# B&R Automation Studio project DancerControl
Automation Studio 4.12.6.106; technology packages: Acp10Arnc0 5.26.1

## Configuration Config1

CPU X20CP1586, AutomationRuntime J4.93, Build 4.1.2, Vc V4.73.2

### Task classes (Cpu.sw)
```
Cyclic#4:
  VMaster <- Axis.VMaster.prg
NcDataObjects: acp10etxen <- Axis.AxisObject.acp10etxen.dob, AxInit <- Axis.AxisObject.RealAxis.AxInit.dob, AcpParTab <- Axis.AxisObject.RealAxis.AcpParTab.dob, VAxInit <- Axis.AxisObject.Virtual.VAxInit.dob
Libraries: Acp10man, Acp10par, NcGlobal, Acp10sim, Acp10_MC, sys_lib, brsystem, runtime, MpAxis, MpBase, MpCom, MTWinder, MTTypes, AsBrMath
```

### Hardware
```
8EIxxxHxD1x.xxxx-1 : 8EIxxxHxD1x.xxxx-1 v2.3.1.1  [PLK1 -> X20CP1586.IF3 (NodeNumber=1) [Cable Type=PowerlinkCable, Length=10, Version=1.0.0.3]]
  MotionTP = Acp10Arnc0
  Simulate = complete
  ActiveMotorSimulation_r1 = on
  BothEndSwitchesAreNormallyOpen_r1 = on
  QuickStopIsNormallyOpen_r1 = on
  ActiveMotorSimulation_r2 = on
  BothEndSwitchesAreNormallyOpen_r2 = on
  QuickStopIsNormallyOpen_r2 = on
X20CP1586 : X20CP1586 v1.10.0.0
  Connector IF2:
    ActivateDevice = 1
  ConfigurationID = DancerControl_Config1
  Simulation = 1
  TimerDeviceType = EPLX2X
  TimerDevice = X20CP1586.IF3
  TaskClassIdleTime = 2000
  FileDevice1
  FileDeviceName1 = USER
  FileDevicePath1 = USER_PATH
```

### Acp10cfg.ncc - X20CP1586/Motion/Acp10cfg.ncc
```
NcConfiguration (Version=5.26.1, NcSwId=Acp10)
  ACP10CF1_typ:
    cnt_nettrc_rec_drive = 1500
    bufsize_trace_upload = 1200
    tc_nc_man_task = Cyclic #1
    glob_pv_as_ncobject = Yes
    ncsys_dl_broadcast = Yes
    ncsys_dl_acp_reset = Yes
    safemc_log_err_to_ax = Yes
    network_init:
      ncsw_init_execute = Yes
      automatic_execute = No
      node_nr_warning = Yes
      net_err_before_ncact = Yes
    nettrc:
      enter_parsecrec = Yes
      enter_ncaction = Yes
      save_ring_startidx = Yes
    cam_prof_download:
      cam_dat_dl_parallel = No
      tc_cam_dl_parallel = Task class for NC Manager task
    plk_if[0]:
      if_name = IF3
      tc_CycDat_PLCopen = Task class for NC Manager task
      mc_broadcast_extdat = No
```

### Acp10map.ncm - X20CP1586/Motion/Acp10map.ncm
```
NcMapping (NcSwId=Acp10, DisabledNodesAreHidden=False)
  NcObject gAxReelA (ModuleId=8EIxxxHxD1x.xxxx-1, Type=ncAXIS, Channel=1, AcoposSimulation=Off, InitParameter=AxInit, AcoposParameter=AcpParTab, Disabled=FALSE, ModuleDisabled=FALSE)
  NcObject gAxReelB (ModuleId=8EIxxxHxD1x.xxxx-1, Type=ncAXIS, Channel=2, AcoposSimulation=Off, InitParameter=AxInit, AcoposParameter=AcpParTab, Disabled=FALSE, ModuleDisabled=FALSE)
  NcObject gVMaster (ModuleId=8EIxxxHxD1x.xxxx-1, Type=ncV_AXIS, Channel=1, InitParameter=VAxInit, Disabled=FALSE, ModuleDisabled=FALSE)
  NcObject 8EIxxxHxD1x.xxxx-1_ncV_AXIS2 (ModuleId=8EIxxxHxD1x.xxxx-1, Type=ncV_AXIS, Channel=2, Disabled=TRUE, ModuleDisabled=FALSE)
```

### Config.mpaxisbasic - X20CP1586/Motion/Config.mpaxisbasic
```
Element gVMasterLink (Type=mpaxisbasic)
  AxisConfiguration = AxisWithConfiguration
    Drive:
      Controller:
        LoopFilters:
          [0]
          [1]
          [2]
Element gReelALink (Type=mpaxisbasic)
  AxisConfiguration = AxisWithConfiguration
    Drive:
      Controller:
        LoopFilters:
          [0]
          [1]
          [2]
Element gReelBLink (Type=mpaxisbasic)
  AxisConfiguration = AxisWithConfiguration
    Drive:
      Controller:
        LoopFilters:
          [0]
          [1]
          [2]
```

## Logical view

Binary libraries used (declarations not repeated): operator, runtime, astime, AsIecCon, Acp10man 5.26.1, Acp10par 5.26.1, NcGlobal 5.26.1, Acp10sim 5.26.1, Acp10_MC 5.26.1, sys_lib, brsystem, MpAxis 1.89.0, MpBase, MpCom 5.24.2, MTWinder, MTTypes, AsBrMath

### Global.typ - Global data types
```iecst
TYPE
	axis_command_typ : 	STRUCT  (*command structure*)
		Power : BOOL; (*switch on the controller*)
		Home : BOOL; (*reference the axis*)
		MoveAbsolute : BOOL; (*move to an defined position*)
		MoveAdditive : BOOL; (*move a defiened distance*)
		MoveVelocity : BOOL; (*start a movement with a defiened velocity*)
		Halt : BOOL; (*stop every active movement*)
		Stop : BOOL; (*stop every active movement as long as is set*)
		MoveJogPos : BOOL; (*move in positive direction as long as is set*)
		MoveJogNeg : BOOL; (*move in negative direction as long as is set*)
		ErrorAcknowledge : BOOL; (*reset active errors*)
		VelocityControl : BOOL; (*activate velocity control*)
	END_STRUCT;
	axis_parameter_typ : 	STRUCT  (*parameter structure*)
		Position : REAL; (*target-position for MoveAbsolute-Command*)
		Distance : REAL; (*distance for MoveAdditive-Command*)
		Velocity : REAL; (*velocity for MoveVelocity-Command*)
		Direction : USINT; (*direction for commanded movements*)
		Acceleration : REAL; (*acceleration for commanded movements*)
		Deceleration : REAL; (*deceleration for commanded movements*)
		HomePosition : REAL; (*target-position for referencing the axis*)
		HomeMode : USINT; (*homing mode*)
		JogVelocity : REAL; (*velocity for jogging movement*)
	END_STRUCT;
	axis_status_typ : 	STRUCT  (*status structure*)
		ErrorID : UINT; (*ErrorID of any occured error*)
		ErrorText : ARRAY[0..3]OF STRING[79]; (*Error Text*)
		ActPosition : REAL; (*actual position of the axis*)
		ActVelocity : REAL; (*actual velocity of the axis*)
		DriveStatus : MpAxisBasicInfoType; (*actual status of the axis*)
		PoweredOn : BOOL; (*Axis powered on *)
		Homed : BOOL; (*Axis Homed*)
	END_STRUCT;
	axis_axisState_typ : 	STRUCT  (*axis state structure*)
		Disabled : BOOL; (*if set, axis is in state Disabled*)
		StandStill : BOOL; (*if set, axis is in state StandsStill*)
		Homing : BOOL; (*if set, axis is in state Homing*)
		Stopping : BOOL; (*if set, axis is in state Stopping*)
		DiscreteMotion : BOOL; (*if set, axis is in state DiscreteMotion*)
		ContinuousMotion : BOOL; (*if set, axis is in state ContinousMotion*)
		SynchronizedMotion : BOOL; (*if set, axis is in state SynchronizedMotion*)
		ErrorStop : BOOL; (*if set, axis is in state ErrorStop*)
	END_STRUCT;
	axis_typ : 	STRUCT  (*control structure*)
		Command : axis_command_typ; (*command structure*)
		Parameter : axis_parameter_typ; (*parameter structure*)
		Status : axis_status_typ; (*status structure*)
		AxisState : axis_axisState_typ; (*axis state structure*)
		Enable : BOOL; (*Axis command enable*)
	END_STRUCT;

END_TYPE
```

### Global.var - Global variables
```iecst
(*Axis Structure *)
VAR
	gAxReelA : ACP10AXIS_typ;
	gAxReelB : ACP10AXIS_typ;
	gVMaster : ACP10VAXIS_typ;
END_VAR
(*Control Axis Structure *)
VAR
	gAxis : ARRAY[0..MAX_AXIS] OF axis_typ;
	AxisIndex : USINT;
END_VAR
```

### Constants.var
```iecst
VAR CONSTANT
	MAX_AXIS : USINT := 3; (*Max value axis to be controlled *)
END_VAR
(*Axis Identifier*)
VAR CONSTANT
	VMASTER : USINT := 0;
	REEL_A : USINT := 1;
	REEL_B : USINT := 2;
	GENERIC : USINT := 3;
END_VAR
(*Axis Parameters*)
VAR CONSTANT
	LINE_ACCELERATION : REAL := 500000.0; (*Acceleration and deceleration of the line axis.*)
	MAX_LINE_DECELERATION : REAL := 1000000.0; (*Maximum deceleration of the line axis.*)
	MAX_DANCER_POSITION : REAL := 500.0; (*Maximum position of the dancer arm.*)
	STANDSTILL_WINDOW : REAL := 0.0; (*Speed dead band*)
	PI : REAL := 3.1416; (*PI Value*)
END_VAR
```


### Program Logical/Axis/VMaster (IEC)

#### Cyclic.st - Cyclic code
```iecst
PROGRAM _CYCLIC

	(**** Call Subroutines ****)
	Act_Main;
	Act_Parameters;

	(** Enable FB's **)
	AxisBasic.Enable 			:= gAxis[AxisIndex].Enable;
	AxisConfig.Enable 		:= AxisBasic.Active;
	ReadAxisError.Enable 	:= AxisBasic.Error OR AxisConfig.Error;

	(**** Definicion sentido de giro del eje ****)
	IF AxisDirection THEN
		Direction	:= mpAXIS_DIR_CLOCKWISE;
	ELSE
		Direction	:= mpAXIS_DIR_COUNTERCLOCKWISE;
	END_IF

	(**** Secuencia configuarcion Eje *****)
	IF NOT ConfigReq THEN
		StConfig := CONFIG_WAIT;
	END_IF

	CASE StConfig OF

		CONFIG_WAIT:

			IF ConfigReq THEN
				StConfig := CONFIG_LOAD_REQ;
			END_IF

		CONFIG_LOAD_REQ:

			(* Carga la configuracion por default en Confing.mpaxisbasic*)
			AxisConfig.Load	:= TRUE;

			IF AxisConfig.CommandDone THEN
				StConfig 			:= CONFIG_LOAD_DONE;
			END_IF

		CONFIG_LOAD_DONE:

			(* Actualiza la configuracion, carga parametros asignados por el usuario *)
			AxisConfig.Load		:= FALSE;
			StConfig 					:= CONFIG_SAVE_REQ;

		CONFIG_SAVE_REQ:

			AxisConfigPar.AxisName 																:= AxisName;

			//Axis

			AxisConfigPar.Axis.BaseType 													:= mpAXIS_PERIODIC_ROTARY;
			AxisConfigPar.Axis.MeasurementUnit 										:= mpAXIS_UNIT_GENERIC;
			AxisConfigPar.Axis.MeasurementResolution 							:= Resolution;
			AxisConfigPar.Axis.PeriodSettings.Period							:= Period;

			AxisConfigPar.Axis.MovementLimits.VelocityPositive		:= LimitSpeed;
			AxisConfigPar.Axis.MovementLimits.VelocityNegative		:= LimitSpeed;
			AxisConfigPar.Axis.MovementLimits.Acceleration				:= LimitAccDec;
			AxisConfigPar.Axis.MovementLimits.Deceleration				:= LimitAccDec;

			//Drive

			AxisConfigPar.Drive.Gearbox.Input											:= GearIn;
			AxisConfigPar.Drive.Gearbox.Output										:= GearOut;
			AxisConfigPar.Drive.Gearbox.Direction 								:= Direction;
			AxisConfigPar.Drive.Transformation.ReferenceDistance 	:= Period;

			(* Salva en el drive los parametros asignados por el usuario *)

			AxisConfig.Save := TRUE;

			IF AxisConfig.CommandDone THEN
				StConfig := CONFIG_SAVE_DONE;
			END_IF

		CONFIG_SAVE_DONE:

			(* Configuracion terminada *)

			AxisConfig.Save := FALSE;
			ConfigReq				:= FALSE;
			ConfigDone			:= TRUE;

	END_CASE

	(********** FB's Configuration *********)

	AxisBasic.Axis 					:= Axis;
	AxisBasic.MpLink 				:= ADR(MpLink);
	AxisBasic.Parameters 		:= ADR(AxisBasicPar);
	AxisBasic();

	AxisConfig.MpLink 			:= ADR(MpLink);
	AxisConfig.Configuration:= ADR(AxisConfigPar);
	AxisConfig();

	ReadAxisError.Axis 			:= Axis;
	ReadAxisError.Mode 			:= mcTEXT;
	ReadAxisError();

	(****************************************)

END_PROGRAM
```

#### Act_Main.st
```iecst
ACTION Act_Main:

	(*Command*)
	gAxis[AxisIndex].Command.Power := AxisBasic.Active AND AxisConfig.Active;
	AxisBasic.Stop := gAxis[AxisIndex].Command.Stop;

	(*Status*)
	gAxis[AxisIndex].Status.ActVelocity := AxisBasic.Velocity;
	gAxis[AxisIndex].Status.ActPosition := LREAL_TO_REAL(AxisBasic.Position);
	gAxis[AxisIndex].Status.PoweredOn 	:= AxisBasic.PowerOn;
	gAxis[AxisIndex].Status.Homed				:= AxisBasic.IsHomed;
	gAxis[AxisIndex].Status.DriveStatus.PLCopenState := AxisBasic.Info.PLCopenState;
	gAxis[AxisIndex].Status.PoweredOn 	:= AxisBasic.PowerOn;

	(*Axis State*)
	gAxis[AxisIndex].AxisState.Disabled 	:= NOT AxisBasic.Active;
	gAxis[AxisIndex].AxisState.StandStill := NOT AxisBasic.MoveActive;
	gAxis[AxisIndex].AxisState.ErrorStop 	:= AxisBasic.Error OR AxisConfig.Error;
	gAxis[AxisIndex].AxisState.StandStill := NOT AxisBasic.MoveActive;
	gAxis[AxisIndex].AxisState.ErrorStop 	:= AxisBasic.Error OR AxisConfig.Error;

	(*Error Reset*)
	IF gAxis[AxisIndex].Command.ErrorAcknowledge THEN
		AxisBasic.ErrorReset := TRUE;
		AxisConfig.ErrorReset := TRUE;
	ELSE
		AxisBasic.ErrorReset := FALSE;
		AxisConfig.ErrorReset := FALSE;
	END_IF

	(**** Configuracion FB Read Axis Error ****)
	ReadAxisError.Configuration.Format 					:= mcWRAP;   //ReadAxisErrorPar;
	ReadAxisError.Configuration.LineLength 			:= SIZEOF(gAxis[AxisIndex].Status.ErrorText[0]);
	ReadAxisError.Configuration.DataLength 			:= SIZEOF(gAxis[AxisIndex].Status.ErrorText);
	ReadAxisError.Configuration.DataAddress 		:= ADR(gAxis[AxisIndex].Status.ErrorText[0]);
	ReadAxisError.Configuration.DataObjectName 	:= 'acp10etxen';

	(**** Error ****)

	IF gAxis[AxisIndex].AxisState.ErrorStop THEN
		StAxis := STATE_ERROR;
	END_IF

	(**** Speed Control/Accel Control ****)

	AxisBasicPar.Velocity 		:= gAxis[AxisIndex].Parameter.Velocity;
	AxisBasicPar.Acceleration	:= gAxis[AxisIndex].Parameter.Acceleration;
	AxisBasicPar.Deceleration := gAxis[AxisIndex].Parameter.Deceleration;

	IF OldVelocity <> AxisBasicPar.Velocity OR OldAccel <> AxisBasicPar.Acceleration OR OldDecel <> AxisBasicPar.Deceleration THEN
		AxisBasic.Update := TRUE;
		OldVelocity := AxisBasicPar.Velocity;
		OldAccel := AxisBasicPar.Acceleration;
		OldDecel := AxisBasicPar.Deceleration;
	ELSE
		AxisBasic.Update := FALSE;
	END_IF

	(**** Checks is the motor is powered On ****)

	IF NOT gAxis[AxisIndex].Command.Power THEN
		StAxis := STATE_WAIT;
	END_IF

	(**** Axis Sequencer ****)

	CASE StAxis OF

		STATE_WAIT:

			IF AxisBasic.Active AND AxisBasic.Info.BootState = mpAXIS_BLP_DONE AND AxisBasic.Info.ReadyToPowerOn AND ConfigDone THEN
				StAxis:= STATE_POWER_ON;
			ELSIF gAxis[AxisIndex].Command.Power AND NOT ConfigDone THEN
				ConfigReq:= TRUE;
			END_IF

		STATE_POWER_ON:

			IF AxisBasic.Info.HardwareInfo.DeviceType = mpAXIS_VIRTUAL THEN
				StAxis:= STATE_HOME;
			END_IF

		STATE_HOME:

			IF NOT AxisBasic.IsHomed THEN
				AxisBasic.Home := TRUE;
			ELSIF AxisBasic.IsHomed THEN
				AxisBasic.Home := FALSE;
				StAxis:= STATE_READY;
			END_IF

		STATE_READY:

			IF gAxis[AxisIndex].Command.MoveVelocity THEN
				StAxis:= STATE_AUTO;
			END_IF

		STATE_AUTO:

			AxisBasic.MoveVelocity := TRUE;

			IF NOT gAxis[AxisIndex].Command.MoveVelocity THEN
				AxisBasic.MoveVelocity := FALSE;
				StAxis:= STATE_STOP;
			END_IF

		STATE_STOP:

			AxisBasic.Stop := TRUE;

			IF AxisBasic.Stopped THEN
				AxisBasic.Stop := FALSE;
				StAxis:= STATE_READY;
			END_IF

		STATE_ERROR :

			AxisBasic.MoveVelocity := FALSE;

			IF gAxis[AxisIndex].Command.ErrorAcknowledge THEN
				StAxis:= STATE_READY;
			END_IF

	END_CASE

	gAxis[AxisIndex].AxisState.ContinuousMotion := StAxis = STATE_AUTO;
	gAxis[AxisIndex].AxisState.Stopping 				:= StAxis = STATE_STOP;
	gAxis[AxisIndex].AxisState.StandStill 			:= StAxis = STATE_READY;

END_ACTION
```

#### Act_Parameters.st
```iecst
ACTION Act_Parameters:

	//---- Numero del Eje ----///
	AxisIndex := VMASTER;

	//---- MpLink ----//
	MpLink 		:= gVMasterLink;
	Axis 			:= ADR(gVMaster);

	//---- Nombre del eje ----//
	AxisName := ' Virtual Master ';

	//---- Hablita el eje ----//
	gAxis[AxisIndex].Enable := TRUE;

	//---- Limite de velocidad -----//
	LimitSpeed 	:= 6600.0;

	//----- Limete de aceleracion/desaceleracion ----//
	LimitAccDec := 6600.0;

	//---- Relacion de velocoidad motor/reductor ----//
	GearIn 	:= 1;
	GearOut := 1;

	//---- Seleccion direccion de rotacion del eje ----//
	AxisDirection := TRUE; // TRUE = sentido de las manesillas del reloj; FALSE = en contra de las manesillas del reloj;

	// ---- Definicion Paramentros de posicion del eje ----//
	Period 				:= 360.0;
	Resolution		:= 0.01;

	/////////////////////////////////////////////////////////////////

END_ACTION
```

#### Init.st - Init code
```iecst
PROGRAM _INIT

	ConfigReq := TRUE;
	Act_Parameters;

END_PROGRAM
```

#### Types.typ - Local data types
```iecst
TYPE
	AxisState_enum :
		( (*Axis control steps*)
		STATE_WAIT := 0,
		STATE_POWER_ON := 10,
		STATE_ERROR := 20,
		STATE_STOP := 30,
		STATE_READY := 40,
		STATE_HOME := 50,
		STATE_AUTO := 60,
		STATE_MANUAL := 70,
		STATE_MAINT := 80
		);
	ConfigStates_enum :
		( (*Axis Configuration steps *)
		CONFIG_WAIT := 0,
		CONFIG_LOAD_REQ := 10,
		CONFIG_LOAD_DONE := 20,
		CONFIG_SAVE_REQ := 30,
		CONFIG_SAVE_DONE := 70,
		CONFIG_COMPLETE := 80
		);
END_TYPE
```

#### Variables.var - Local variables
```iecst
	(*Mp Axis FB*)
VAR
		AxisBasic : MpAxisBasic;
		AxisBasicPar : MpAxisBasicParType;
		AxisConfig : MpAxisBasicConfig;
		AxisConfigPar : MpAxisBasicConfigType;
		ReadAxisError : MC_BR_ReadAxisError;
END_VAR
	(*Axis Control Var *)
	VAR
		Axis : UDINT; (*Axis*)
		AxisIndex : USINT; (*Axis Index *)
		StAxis : AxisState_enum; (*Axis control steps*)
		MpLink : MpComIdentType; (*Axis basic parameters structure*)
END_VAR
	(*Axis Speed Control var *)
	VAR
		OldVelocity : REAL; (*Old Velocity Value*)
END_VAR
	(*Axis Configuration*)
	VAR
		StConfig : ConfigStates_enum; (*Configuration steps*)
		ConfigDone : BOOL; (*Configuration done*)
		AxisDirection : BOOL; (*Command direction 1 = CW; 0 = CCW*)
		Direction : MpAxisMotorDirectionEnum; (*Status diection *)
		ConfigReq : BOOL; (*Configuration command*)
		LimitSpeed : REAL; (*Speed limmit*)
		LimitAccDec : REAL; (*acceleratio/Deceleration limit*)
		GearIn : UDINT; (*Input ratio*)
		GearOut : UDINT; (*output ratio*)
		Period : LREAL; (*Period  exemple 360.0 degrees.*)
		Resolution : REAL; (*Minimum distance that can be used for a movement*)
		AxisName : STRING[20]; (*Axis Name *)
		OldAccel : REAL; (*Old Acel value *)
		OldDecel : REAL; (*Old  decel value*)
END_VAR
```

### Data object Logical/Axis/AxisObject/acp10etxen (Ett)

- acp10etxen.ett (not shown)

### Program Logical/Axis/ReelA

#### Types.typ
```iecst
TYPE
	AxisState_enum :
		( (*Axis control steps*)
		STATE_WAIT := 0,
		STATE_POWER_ON := 10,
		STATE_ERROR := 20,
		STATE_STOP := 30,
		STATE_READY := 40,
		STATE_HOME := 50,
		STATE_AUTO := 60,
		STATE_MANUAL := 70,
		STATE_MAINT := 80
	);
	ConfigStates_enum :
		( (*Axis Configuration steps *)
		CONFIG_WAIT := 0,
		CONFIG_LOAD_REQ := 10,
		CONFIG_LOAD_DONE := 20,
		CONFIG_SAVE_REQ := 30,
		CONFIG_SAVE_DONE := 70
	);

END_TYPE
```

#### Variables.var
```iecst
VAR
	(*Mp Axis FB*)
	AxisBasic : MpAxisBasic;
	AxisBasicPar : MpAxisBasicParType;
	AxisConfig : MpAxisBasicConfig;
	AxisConfigPar : MpAxisBasicConfigType;
	ReadAxisError : MC_BR_ReadAxisError;
	VelocityControl : MC_BR_VelocityControl; (*Function Block*)
END_VAR
(*Axis Control Var *)
VAR
	Axis : UDINT;(*Axis*)
	AxisIndex : USINT; (*Axis Index *)
	StAxis : AxisState_enum; (*Axis control steps*)
	MpLink : MpComIdentType;  (*Axis basic parameters structure*)
END_VAR
(*Axis Speed Control var *)
VAR
	OldVelocity : REAL; (*Old Velocity Value*)
END_VAR
(*Axis Configuration*)
VAR
	StConfig : ConfigStates_enum; (*Configuration steps*)
	ConfigDone : BOOL;(*Configuration done*)
	AxisDirection : BOOL; (*Command direction 1 = CW; 0 = CCW*)
	Direction : MpAxisMotorDirectionEnum; (*Status diection *)
	ConfigReq : BOOL; (*Configuration command*)
	LimitSpeed : REAL;(*Speed limmit*)
	LimitAccDec : REAL;(*acceleratio/Deceleration limit*)
	GearIn : UDINT;
	GearOut : UDINT;
	Period : LREAL;
	Resolution : REAL;
	AxisName : STRING[20];
END_VAR
```

#### Act_Main.st
```iecst
ACTION Act_Main:

	(*Command*)
	gAxis[AxisIndex].Command.Power := AxisBasic.Active AND AxisConfig.Active;
	AxisBasic.Stop := gAxis[AxisIndex].Command.Stop;

	(*Status*)
	gAxis[AxisIndex].Status.ActVelocity := AxisBasic.Velocity;
	gAxis[AxisIndex].Status.ActPosition := LREAL_TO_REAL(AxisBasic.Position);
	gAxis[AxisIndex].Status.PoweredOn 	:= AxisBasic.PowerOn;
	gAxis[AxisIndex].Status.Homed				:= AxisBasic.IsHomed;
	gAxis[AxisIndex].Status.DriveStatus.PLCopenState := AxisBasic.Info.PLCopenState;
	gAxis[AxisIndex].Status.PoweredOn 	:= AxisBasic.PowerOn;

	(*Axis State*)
	gAxis[AxisIndex].AxisState.Disabled 	:= NOT AxisBasic.Active;
	gAxis[AxisIndex].AxisState.StandStill := NOT AxisBasic.MoveActive;
	gAxis[AxisIndex].AxisState.ErrorStop 	:= AxisBasic.Error OR AxisConfig.Error;
	gAxis[AxisIndex].AxisState.StandStill := NOT AxisBasic.MoveActive;
	gAxis[AxisIndex].AxisState.ErrorStop 	:= AxisBasic.Error OR AxisConfig.Error;

	(*Error Reset*)
	IF gAxis[AxisIndex].Command.ErrorAcknowledge THEN
		AxisBasic.ErrorReset := TRUE;
		AxisConfig.ErrorReset := TRUE;
	ELSE
		AxisBasic.ErrorReset := FALSE;
		AxisConfig.ErrorReset := FALSE;
	END_IF

	(**** Configuracion FB Read Axis Error ****)
	ReadAxisError.Configuration.Format 					:= mcWRAP;   //ReadAxisErrorPar;
	ReadAxisError.Configuration.LineLength 			:= SIZEOF(gAxis[AxisIndex].Status.ErrorText[0]);
	ReadAxisError.Configuration.DataLength 			:= SIZEOF(gAxis[AxisIndex].Status.ErrorText);
	ReadAxisError.Configuration.DataAddress 		:= ADR(gAxis[AxisIndex].Status.ErrorText[0]);
	ReadAxisError.Configuration.DataObjectName 	:= 'acp10etxen';

	(**** Error ****)

	IF gAxis[AxisIndex].AxisState.ErrorStop THEN
		StAxis := STATE_ERROR;
	END_IF

//	(**** Speed Control/Accel Control ****)
//
//	AxisBasicPar.Velocity 		:= gAxis[AxisIndex].Parameter.Velocity;
//	AxisBasicPar.Acceleration	:= gAxis[AxisIndex].Parameter.Acceleration;
//	AxisBasicPar.Deceleration := gAxis[AxisIndex].Parameter.Deceleration;
//
//	IF OldVelocity <> AxisBasicPar.Velocity OR OldAccel <> AxisBasicPar.Acceleration OR OldDecel <> AxisBasicPar.Deceleration THEN
//		AxisBasic.Update := TRUE;
//		OldVelocity := AxisBasicPar.Velocity;
//		OldAccel := AxisBasicPar.Acceleration;
//		OldDecel := AxisBasicPar.Deceleration;
//	ELSE
//		AxisBasic.Update := FALSE;
//	END_IF

	(**** Checks is the motor is powered On ****)

	IF NOT gAxis[AxisIndex].Command.Power THEN
		StAxis := STATE_WAIT;
	END_IF

	(**** Checks the motor error ****)

	IF gAxis[AxisIndex].AxisState.ErrorStop THEN
		StAxis:= STATE_ERROR;
	END_IF

	(**** Axis Sequencer ****)

	CASE StAxis OF

		STATE_WAIT:

			IF AxisBasic.Active AND AxisBasic.Info.BootState = mpAXIS_BLP_DONE AND AxisConfig.Active AND AxisBasic.Info.ReadyToPowerOn AND ConfigDone THEN
				StAxis:= STATE_POWER_ON;
			ELSIF gAxis[AxisIndex].Command.Power AND NOT ConfigDone THEN
				ConfigReq:= TRUE;
			END_IF

		STATE_POWER_ON:

			IF gAxis[AxisIndex].Command.Power AND NOT AxisBasic.PowerOn THEN
				AxisBasic.Power := TRUE;
			ELSIF AxisBasic.PowerOn THEN
				StAxis:= STATE_HOME;
			END_IF

		STATE_HOME:

			IF NOT AxisBasic.IsHomed THEN
				AxisBasic.Home := TRUE;
			ELSIF AxisBasic.IsHomed THEN
				AxisBasic.Home := FALSE;
				StAxis:= STATE_READY;
			END_IF

		STATE_READY:

			IF gAxis[AxisIndex].Command.VelocityControl THEN
				StAxis:= STATE_AUTO;
			END_IF

		STATE_AUTO:

			(******************** VELOCITY CONTROL **********************)
			(* STATE: velocity control *)
			(* activate MC_BR_VelocityControl *)
						VelocityControl.Enable := TRUE;
						VelocityControl.CyclicVelocity := gSetWinderVelocity;
						VelocityControl.CyclicVelocityCorrection :=  gVelocityCorrection;
						VelocityControl.CyclicTorque := gSetMotorTorque;
						VelocityControl.Acceleration := gAxis[AxisIndex].Parameter.Acceleration;
						VelocityControl.Deceleration := gAxis[AxisIndex].Parameter.Deceleration ;
						VelocityControl.TorqueMode := mcFF;
						VelocityControl.SctrlKv := gActProportionalGain;
						VelocityControl.SctrlTn := gActIntegrationTime;
			(* this feature is not possible for ACOPOS simulation *)
			// VelocityControl.InitSctrl := gControl.Winder.InitSpeedController;

			IF NOT gAxis[AxisIndex].Command.VelocityControl THEN
				VelocityControl.Enable := FALSE;
				StAxis:= STATE_READY;
			END_IF

		STATE_ERROR:

			VelocityControl.Enable := FALSE;

	END_CASE

END_ACTION
```

#### Act_Parameters.st
```iecst
ACTION Act_Parameters:

	//---- Numero del Eje ----///
	AxisIndex := REEL_A;

	//---- MpLink ----//
	MpLink 		:= gReelALink;
	Axis 			:= ADR(gAxReelA);

	//---- Nombre del eje ----//
	AxisName := ' Reel A ';

	//---- Hablita el eje ----//
	gAxis[AxisIndex].Enable := TRUE;

	//---- Limite de velocidad -----//
	LimitSpeed 	:= 6600.0;

	//----- Limete de aceleracion/desaceleracion ----//
	LimitAccDec := 6600.0;

	//---- Relacion de velocoidad motor/reductor ----//
	GearIn 	:= 1;
	GearOut := 1;

	//---- Seleccion direccion de rotacion del eje ----//
	AxisDirection := TRUE; // TRUE = sentido de las manesillas del reloj; FALSE = en contra de las manesillas del reloj;

	// ---- Definicion Paramentros de posicion del eje ----//
	Period 				:= 360.0;
	Resolution		:= 0.001;

	/////////////////////////////////////////////////////////////////

END_ACTION
```

#### Cyclic.st
```iecst
PROGRAM _CYCLIC

(**** Call Subroutines ****)
	Act_Main;
	Act_Parameters;

	(** Enable FB's **)
	AxisBasic.Enable 			:= gAxis[AxisIndex].Enable;
	AxisConfig.Enable 		:= AxisBasic.Active;
	ReadAxisError.Enable 	:= AxisBasic.Error OR AxisConfig.Error;

	(**** Definicion sentido de giro del eje ****)
	IF AxisDirection THEN
		Direction	:= mpAXIS_DIR_CLOCKWISE;
	ELSE
		Direction	:= mpAXIS_DIR_COUNTERCLOCKWISE;
	END_IF

	(**** Secuencia configuarcion Eje *****)
	IF NOT ConfigReq THEN
		StConfig := CONFIG_WAIT;
	END_IF

	CASE StConfig OF

		CONFIG_WAIT:

			IF ConfigReq THEN
				StConfig := CONFIG_LOAD_REQ;
			END_IF

		CONFIG_LOAD_REQ:

			(* Carga la configuracion por default en Confing.mpaxisbasic*)
			AxisConfig.Load	:= TRUE;

			IF AxisConfig.CommandDone THEN
				StConfig 			:= CONFIG_LOAD_DONE;
			END_IF

		CONFIG_LOAD_DONE:

			(* Actualiza la configuracion, carga parametros asignados por el usuario *)
			AxisConfig.Load		:= FALSE;
			StConfig 					:= CONFIG_SAVE_REQ;

		CONFIG_SAVE_REQ:

			AxisConfigPar.AxisName 																:= AxisName;

			//Axis

			AxisConfigPar.Axis.BaseType 													:= mpAXIS_PERIODIC_ROTARY;
			AxisConfigPar.Axis.MeasurementUnit 										:= mpAXIS_UNIT_GENERIC;
			AxisConfigPar.Axis.MeasurementResolution 							:= Resolution;
			AxisConfigPar.Axis.PeriodSettings.Period							:= Period;

			AxisConfigPar.Axis.MovementLimits.VelocityPositive		:= LimitSpeed;
			AxisConfigPar.Axis.MovementLimits.VelocityNegative		:= LimitSpeed;
			AxisConfigPar.Axis.MovementLimits.Acceleration				:= LimitAccDec;
			AxisConfigPar.Axis.MovementLimits.Deceleration				:= LimitAccDec;

			//Drive

			AxisConfigPar.Drive.Gearbox.Input											:= GearIn;
			AxisConfigPar.Drive.Gearbox.Output										:= GearOut;
			AxisConfigPar.Drive.Gearbox.Direction 								:= Direction;
			AxisConfigPar.Drive.Transformation.ReferenceDistance 	:= Period;

			(* Salva en el drive los parametros asignados por el usuario *)

			AxisConfig.Save := TRUE;

			IF AxisConfig.CommandDone THEN
				StConfig := CONFIG_SAVE_DONE;
			END_IF

		CONFIG_SAVE_DONE:

			(* Configuracion terminada *)

			AxisConfig.Save := FALSE;
			ConfigReq				:= FALSE;
			ConfigDone			:= TRUE;

	END_CASE

	(********** FB's Configuration *********)

	AxisBasic.Axis 					:= Axis;
	AxisBasic.MpLink 				:= ADR(MpLink);
	AxisBasic.Parameters 		:= ADR(AxisBasicPar);
	AxisBasic();

	AxisConfig.MpLink 			:= ADR(MpLink);
	AxisConfig.Configuration:= ADR(AxisConfigPar);
	AxisConfig();

	ReadAxisError.Axis 			:= Axis;
	ReadAxisError.Mode 			:= mcTEXT;
	ReadAxisError();

	VelocityControl();
	(****************************************)

END_PROGRAM
```

### Program Logical/Axis/ReelB

#### Types.typ
```iecst
TYPE
	AxisState_enum :
		( (*Axis control steps*)
		STATE_WAIT := 0,
		STATE_POWER_ON := 10,
		STATE_ERROR := 20,
		STATE_STOP := 30,
		STATE_READY := 40,
		STATE_HOME := 50,
		STATE_AUTO := 60,
		STATE_MANUAL := 70,
		STATE_MAINT := 80
	);
	ConfigStates_enum :
		( (*Axis Configuration steps *)
		CONFIG_WAIT := 0,
		CONFIG_LOAD_REQ := 10,
		CONFIG_LOAD_DONE := 20,
		CONFIG_SAVE_REQ := 30,
		CONFIG_SAVE_DONE := 70
	);
END_TYPE
```

#### Variables.var
```iecst
VAR
	(*Mp Axis FB*)
	AxisBasic : MpAxisBasic;
	AxisBasicPar : MpAxisBasicParType;
	AxisConfig : MpAxisBasicConfig;
	AxisConfigPar : MpAxisBasicConfigType;
	ReadAxisError : MC_BR_ReadAxisError;
	VelocityControl : MC_BR_VelocityControl; (*Function Block*)
END_VAR
(*Axis Control Var *)
VAR
	Axis : UDINT;(*Axis*)
	AxisIndex : USINT; (*Axis Index *)
	StAxis : AxisState_enum; (*Axis control steps*)
	MpLink : MpComIdentType;  (*Axis basic parameters structure*)
END_VAR
(*Axis Speed Control var *)
VAR
	OldVelocity : REAL; (*Old Velocity Value*)
END_VAR
(*Axis Configuration*)
VAR
	StConfig : ConfigStates_enum; (*Configuration steps*)
	ConfigDone : BOOL;(*Configuration done*)
	AxisDirection : BOOL; (*Command direction 1 = CW; 0 = CCW*)
	Direction : MpAxisMotorDirectionEnum; (*Status diection *)
	ConfigReq : BOOL; (*Configuration command*)
	LimitSpeed : REAL;(*Speed limmit*)
	LimitAccDec : REAL;(*acceleratio/Deceleration limit*)
	GearIn : UDINT;
	GearOut : UDINT;
	Period : LREAL;
	Resolution : REAL;
	AxisName : STRING[20];
END_VAR
```

#### Act_Parameters.st
```iecst
ACTION Act_Parameters:

	//---- Numero del Eje ----///
	AxisIndex := REEL_B;

	//---- MpLink ----//
	MpLink 		:= gReelBLink;
	Axis 			:= ADR(gAxReelB);

	//---- Nombre del eje ----//
	AxisName := ' Reel A ';

	//---- Hablita el eje ----//
	gAxis[AxisIndex].Enable := TRUE;

	//---- Limite de velocidad -----//
	LimitSpeed 	:= 6600.0;

	//----- Limete de aceleracion/desaceleracion ----//
	LimitAccDec := 6600.0;

	//---- Relacion de velocoidad motor/reductor ----//
	GearIn 	:= 1;
	GearOut := 1;

	//---- Seleccion direccion de rotacion del eje ----//
	AxisDirection := TRUE; // TRUE = sentido de las manesillas del reloj; FALSE = en contra de las manesillas del reloj;

	// ---- Definicion Paramentros de posicion del eje ----//
	Period 				:= 360.0;
	Resolution		:= 0.001;

	/////////////////////////////////////////////////////////////////

END_ACTION
```

#### Cyclic.st
```iecst
PROGRAM _CYCLIC

	(**** Call Subroutines ****)
	Act_Main;
	Act_Parameters;

	(** Enable FB's **)
	AxisBasic.Enable 			:= gAxis[AxisIndex].Enable;
	AxisConfig.Enable 		:= AxisBasic.Active;
	ReadAxisError.Enable 	:= AxisBasic.Error OR AxisConfig.Error;

	(**** Definicion sentido de giro del eje ****)
	IF AxisDirection THEN
		Direction	:= mpAXIS_DIR_CLOCKWISE;
	ELSE
		Direction	:= mpAXIS_DIR_COUNTERCLOCKWISE;
	END_IF

	(**** Secuencia configuarcion Eje *****)
	IF NOT ConfigReq THEN
		StConfig := CONFIG_WAIT;
	END_IF

	CASE StConfig OF

		CONFIG_WAIT:

			IF ConfigReq THEN
				StConfig := CONFIG_LOAD_REQ;
			END_IF

		CONFIG_LOAD_REQ:

			(* Carga la configuracion por default en Confing.mpaxisbasic*)
			AxisConfig.Load	:= TRUE;

			IF AxisConfig.CommandDone THEN
				StConfig 			:= CONFIG_LOAD_DONE;
			END_IF

		CONFIG_LOAD_DONE:

			(* Actualiza la configuracion, carga parametros asignados por el usuario *)
			AxisConfig.Load		:= FALSE;
			StConfig 					:= CONFIG_SAVE_REQ;

		CONFIG_SAVE_REQ:

			AxisConfigPar.AxisName 																:= AxisName;

			//Axis

			AxisConfigPar.Axis.BaseType 													:= mpAXIS_PERIODIC_ROTARY;
			AxisConfigPar.Axis.MeasurementUnit 										:= mpAXIS_UNIT_GENERIC;
			AxisConfigPar.Axis.MeasurementResolution 							:= Resolution;
			AxisConfigPar.Axis.PeriodSettings.Period							:= Period;

			AxisConfigPar.Axis.MovementLimits.VelocityPositive		:= LimitSpeed;
			AxisConfigPar.Axis.MovementLimits.VelocityNegative		:= LimitSpeed;
			AxisConfigPar.Axis.MovementLimits.Acceleration				:= LimitAccDec;
			AxisConfigPar.Axis.MovementLimits.Deceleration				:= LimitAccDec;

			//Drive

			AxisConfigPar.Drive.Gearbox.Input											:= GearIn;
			AxisConfigPar.Drive.Gearbox.Output										:= GearOut;
			AxisConfigPar.Drive.Gearbox.Direction 								:= Direction;
			AxisConfigPar.Drive.Transformation.ReferenceDistance 	:= Period;

			(* Salva en el drive los parametros asignados por el usuario *)

			AxisConfig.Save := TRUE;

			IF AxisConfig.CommandDone THEN
				StConfig := CONFIG_SAVE_DONE;
			END_IF

		CONFIG_SAVE_DONE:

			(* Configuracion terminada *)

			AxisConfig.Save := FALSE;
			ConfigReq				:= FALSE;
			ConfigDone			:= TRUE;

	END_CASE

	(********** FB's Configuration *********)

	AxisBasic.Axis 					:= Axis;
	AxisBasic.MpLink 				:= ADR(MpLink);
	AxisBasic.Parameters 		:= ADR(AxisBasicPar);
	AxisBasic();

	AxisConfig.MpLink 			:= ADR(MpLink);
	AxisConfig.Configuration:= ADR(AxisConfigPar);
	AxisConfig();

	ReadAxisError.Axis 			:= Axis;
	ReadAxisError.Mode 			:= mcTEXT;
	ReadAxisError();

	VelocityControl();
	(****************************************)

END_PROGRAM
```

#### Init.st
```iecst
PROGRAM _INIT

	ConfigReq := TRUE;
	Act_Parameters;

END_PROGRAM
```

### Program Logical/DancerCtrl/LineCtrl (IEC)

#### Types.typ
```iecst
TYPE
	AxisState_enum :
		( (*States*)
		STATE_HOMING, (*Homing axis*)
		STATE_STANDSTILL, (*Axis ready*)
		STATE_MOTION, (*Continious movement*)
		STATE_STOPPING (*Stopping*)
	);
END_TYPE
```

#### Variables.var
```iecst
VAR
	RollerDiamter : REAL;
	LinearVelocity : REAL;
	AngularVelocity : REAL;
	Start : BOOL;
	StLineCtrl : AxisState_enum;
	Stop : BOOL;
END_VAR
```

#### Main.st
```iecst
PROGRAM _INIT

	(**** Datos de simulacion ****)
	RollerDiamter:= 100.0; // Diametro del rodillo en milimetros
	gAxis[VMASTER].Parameter.Acceleration := 10000.0; // grados/s
	gAxis[VMASTER].Parameter.Deceleration := 10000.0; // grados/s
	LinearVelocity := 400.0; // Setpoint en mm/s

END_PROGRAM

PROGRAM _CYCLIC

	(**** Calculo de velocidad para cambiarla a mm/s ****)
	gAxis[VMASTER].Parameter.Velocity := ((LinearVelocity * 360)/(PI * RollerDiamter));
	AngularVelocity := (gAxis[VMASTER].Status.ActVelocity * (PI/180)) * (RollerDiamter / 2);
	(*LinearVelocity := gControl.Cmd.LineVelocity;*)
	gLineVelocity :=  AngularVelocity/0.001;

	CASE StLineCtrl OF

		STATE_HOMING:

			(*************** STATE HOMING **************************)

			IF gAxis[VMASTER].Status.Homed THEN
				StLineCtrl:= STATE_STANDSTILL;
			END_IF

		STATE_STANDSTILL:

			(*************** STATE STANDSTILL **********************)

			IF Start THEN
				StLineCtrl := STATE_MOTION;
			END_IF

		STATE_MOTION:

			(*************** STATE MOTION **************************)

			(*gAxis[VMASTER].Parameter.Acceleration := 10000.0; // grados/s*)
			(*gAxis[VMASTER].Parameter.Deceleration := 10000.0; // grados/s*)

			Start := FALSE;
			gAxis[VMASTER].Command.MoveVelocity := TRUE;
			gAxis[REEL_A].Command.VelocityControl := TRUE;

			IF Stop THEN
				gAxis[VMASTER].Command.MoveVelocity := FALSE;
				gAxis[REEL_A].Command.VelocityControl := FALSE;
				StLineCtrl := STATE_STOPPING;
			END_IF

		STATE_STOPPING:

			(*************** STATE STOPPING ************************)

			Stop := FALSE;

			IF gAxis[VMASTER].Status.ActVelocity = 0.0 THEN
				StLineCtrl:= STATE_STANDSTILL;
			END_IF

	END_CASE

END_PROGRAM

PROGRAM _EXIT
	(* Insert code here *)

END_PROGRAM
```

### Program Logical/DancerCtrl/DancerController (IEC)

#### Cyclic.st - Cyclic code
```iecst
PROGRAM _CYCLIC

	Act_DiamEstimator;
	Act_Dancer;
	Act_SimModel;
	Act_AxisController;

END_PROGRAM
```

#### Act_DiamEstimator.st
```iecst
ACTION Act_DiamEstimator:

	DiameterEstimator.ActLinePosition := ActLinePosition;
	DiameterEstimator.ActWinderPosition := ActWinderPosition;
	DiameterEstimator.ActDancerPosition := ActDancerPosition;

	ActDiameter := DiameterEstimator.ActDiameter;

	(*************** DiameterEstimator ***********************)

	ActLinePosition		:= REAL_TO_DINT(gAxis[VMASTER].Status.ActPosition);
	ActWinderPosition := REAL_TO_DINT(gAxis[REEL_A].Status.ActPosition);

	DiameterEstimator();

END_ACTION
```

#### Act_Dancer.st
```iecst
ACTION Act_Dancer:

	DancerController.SetDancerPosition := SetDancerPosition;
	DancerController.ActDancerPosition := ActDancerPosition;

	DancerController.ActDiameter := ActDiameter;

	(*************** DancerController *************************)

	DancerController();

	VelocityCorrection := DancerController.VelocityCorrection;

	gVelocityCorrection := VelocityCorrection;

END_ACTION
```

#### Act_SimModel.st
```iecst
ACTION Act_SimModel:

	SimulationModel.Configuration := ConfigurationParameters;
	SimulationModel.Parameters := SimulationParameters;
	SimulationModel.SetLineVelocity := SetLineVelocity;

	SimulationModel.SetWinderVelocity := SetWinderVelocity;
	SimulationModel.WinderVelocityCorrection := WinderVelocityCorrection;
	SimulationModel.SetMotorTorque := SetMotorTorque;

	SimulationModel.ActProportionalGain := ActProportionalGain;
	SimulationModel.ActIntegrationTime := ActIntegrationTime;
	SimulationModel.InitSpeedController := InitSpeedController;

	(*************** SimulationModel **************************)

	SimulationModel();

END_ACTION
```

#### Act_AxisController.st
```iecst
ACTION Act_AxisController:

	SetLineVelocity := gLineVelocity; // Noe

	AxisController.SetLineVelocity  :=  SetLineVelocity;
	AxisController.ActDiameter  :=  ActDiameter;
	AxisController.SetMaterialTension  :=  SetMaterialTension;

	AxisController.SynchronizationTime  :=  SynchronistionTime;
	AxisController.StartSynchronization  :=  StartSynchronisation;
	AxisController.StopSynchronization  :=  StopSynchronisation;

	AxisController();

	SetWinderVelocity  :=  AxisController.SetWinderVelocity;
	SetMotorTorque  :=  AxisController.SetMotorTorque;

	ActProportionalGain  :=  AxisController.ActProportionalGain;
	ActIntegrationTime  :=  AxisController.ActIntegrationTime;
	InitSpeedController  :=  AxisController.InitSpeedController;

	gSetWinderVelocity := SetWinderVelocity;
	gSetMotorTorque := SetMotorTorque;
	gActProportionalGain := ActProportionalGain;
	gActIntegrationTime := ActIntegrationTime;
	gInitSpeedController := InitSpeedController;
END_ACTION
```

#### Init.st - Init code
```iecst
PROGRAM _INIT
	(*Simulation*)
	SimulationModel.Enable := TRUE;

	ConfigurationParameters.Geometry.WinderWidth := 1000.0;
	ConfigurationParameters.Geometry.MaterialThickness := 80.0;
	ConfigurationParameters.Geometry.MaxDiameter := 900.0;
	ConfigurationParameters.Geometry.MinDiameter := 90.0;
	ConfigurationParameters.Geometry.MinInertia := 0.39;
	ConfigurationParameters.Geometry.TestDiameter := 820.6;
	ConfigurationParameters.Geometry.TestInertia := 4.3;

	ConfigurationParameters.Axis.LineUnits := 100000; (* 1 (line) unit = =  1 µm *)
	ConfigurationParameters.Axis.WinderUnits := 360000;    (* 1 winder (unit) = =  0.001° *)
	ConfigurationParameters.Axis.RevMotor := 25;
	ConfigurationParameters.Axis.GearRatio := 2.5; (* gear ratio [1] *)
	ConfigurationParameters.Axis.WinderType := mtWND_UNWIND; (* unwinder *)

	SimulationParameters.MaterialLength := 4000.0;
	SimulationParameters.StartDiameter := 820.2;
	SimulationParameters.DancerInertia := 3.25;
	SimulationParameters.DancerLength := 500.0;
	SimulationParameters.MaxDancerPosition := 240.0;
	SimulationParameters.SpeedTorqueFactor := 0.01;
	SimulationParameters.TorqueConstant := 2.1;
	SimulationParameters.Noise := 1; (* additive noise *)
	SimulationModel.ModelType := mtWND_DANCER;
	SimulationModel.TorqueMode := mtWND_TORQUE_FF;
	SimulationModel.SetDancerTorque := 200.0;

	InitSpeedController := TRUE;
	ActProportionalGain := 88.6;
	ActIntegrationTime := 0.143;

	(*Diameter Estimation*)
	DiameterEstimator.Enable := TRUE;

	DiameterEstimator.Configuration.Geometry.WinderWidth := 1000; (*mm*)
	DiameterEstimator.Configuration.Geometry.MaterialThickness := 80.0; (*µm*)
	DiameterEstimator.Configuration.Geometry.MaxDiameter := 900.0; (*mm*)
	DiameterEstimator.Configuration.Geometry.MinDiameter := 90.0; (*mm*)
	DiameterEstimator.Configuration.Geometry.MinInertia := 0.39; (*kgm²*)
	DiameterEstimator.Configuration.Geometry.TestDiameter := 820.6;
	DiameterEstimator.Configuration.Geometry.TestInertia := 4.30;

	DiameterEstimator.Configuration.Axis.LineUnits := 1000000; (* 1 (line) unit := :=  1 µm *)
	DiameterEstimator.Configuration.Axis.WinderUnits := 360000; (* 1 winder (unit) := :=  0.001° *)
	DiameterEstimator.Configuration.Axis.RevMotor := 1;
	DiameterEstimator.Configuration.Axis.GearRatio := 1.0; (* gear ratio := 1 *)
	DiameterEstimator.Configuration.Axis.WinderType := mtWND_UNWIND; (* unwinding system *)

	DiameterEstimator.Parameters.CyclicEstimationWindow := 360000;

	DiameterEstimator.Mode := mtWND_POSITION_BASED;

	(*Dancer*)
	DancerController.Enable := TRUE;

	DancerController.Configuration.Geometry.WinderWidth := 1000;
	DancerController.Configuration.Geometry.MaterialThickness := 80.0;
	DancerController.Configuration.Geometry.MaxDiameter := 900.0;
	DancerController.Configuration.Geometry.MinDiameter := 90.0;
	DancerController.Configuration.Geometry.MinInertia := 0.39;
	DancerController.Configuration.Geometry.TestDiameter := 820.6;
	DancerController.Configuration.Geometry.TestInertia := 4.30;

	DancerController.Configuration.Axis.LineUnits := 1000000; (* 1 (line) unit == 1 µm *)
	DancerController.Configuration.Axis.WinderUnits := 360000; (* 1 winder (unit) == 0.001° *)
	DancerController.Configuration.Axis.RevMotor := 1;
	DancerController.Configuration.Axis.GearRatio := 1.0; (* gear ratio = 1 *)
	DancerController.Configuration.Axis.WinderType := mtWND_UNWIND; (* unwinding system *)

	DancerController.Parameters.PIDParameters.Gain := 2.0;
	DancerController.Parameters.PIDParameters.IntegrationTime := 1.0;
	DancerController.Parameters.PIDParameters.DerivativeTime := 0.0;
	DancerController.Parameters.PIDParameters.FilterTime := 0.0;
	DancerController.Parameters.MaxLineVelocityCorrection := 1000.0; (* == 1 m/s *)
	DancerController.Parameters.MaxControlError := 0.0; (* material break detection off *)

	SetDancerPosition := 150.0;
	ActDiameter := 895.7;

	(*Axis Controller*)
	AxisController.Enable  :=  TRUE;

	AxisController.Configuration.Geometry.WinderWidth  :=  1000;
	AxisController.Configuration.Geometry.MaterialThickness  :=  80.0;
	AxisController.Configuration.Geometry.MaxDiameter  :=  900.0;
	AxisController.Configuration.Geometry.MinDiameter  :=  90.0;
	AxisController.Configuration.Geometry.MinInertia  :=  0.39;
	AxisController.Configuration.Geometry.TestDiameter  :=  820.6;
	AxisController.Configuration.Geometry.TestInertia  :=  4.30;

	AxisController.Configuration.Axis.LineUnits  :=  1000000; (* 1 (line) unit  :=  :=  1 µm *)
	AxisController.Configuration.Axis.WinderUnits  :=  360000; (* 1 winder (unit)  :=  :=  0.001° *)
	AxisController.Configuration.Axis.RevMotor  :=  1;
	AxisController.Configuration.Axis.GearRatio  :=  1.0; (* gear ratio  :=  1 *)
	AxisController.Configuration.Axis.WinderType  :=  mtWND_UNWIND; (* unwinding system *)

	AxisController.Parameters.MinTorque  :=  -50.0;
	AxisController.Parameters.MaxTorque  :=  50.0;

	AxisController.Parameters.Interpolation.MinProportionalGain  :=  20.6;
	AxisController.Parameters.Interpolation.TestProportionalGain  :=  88.6;
	AxisController.Parameters.Interpolation.MinIntegrationTime  :=  0.043;
	AxisController.Parameters.Interpolation.TestIntegrationTime  :=  0.143;

	//ActDiameter  :=  895.7;
	ActInertia  :=  4.7;
	SetMaterialTension  :=  150.0;

END_PROGRAM
```

#### Variables.var - Local variables
```iecst
(*Winder Diameter Estimation*)
VAR
	DiameterEstimator : MTWinderDiameterEstimator; (*diameter estimator*)
	ActLinePosition : DINT; (*actual line position*)
	ActWinderPosition : DINT; (*actual winder position*)
	ActDancerPosition : REAL; (*actual dancer position*)
END_VAR
(* Dancer Controller *)
VAR
	DancerController : MTWinderDancerController; (*tension controller*)
	SetDancerPosition : REAL; (*set material tension*)
	ActDiameter : REAL; (*actual diameter*)
	VelocityCorrection : REAL; (*actual velocity correction*)
END_VAR
(*Simulation Model*)
VAR
	ConfigurationParameters : MTWinderConfigurationType; (* configuration parameters *)
	SimulationParameters : MTWinderSimulationModelType; (* simulation model parameters *)
	SetLineVelocity : REAL; (* set line velocity *)
	SetWinderVelocity : REAL; (* set winder velocity *)
	WinderVelocityCorrection : REAL; (* winder velocity correction *)
	SetMotorTorque : REAL; (* set motor torque *)
	ActProportionalGain : REAL; (* proportional gain *)
	ActIntegrationTime : REAL; (* integration time *)
	InitSpeedController : BOOL; (* initialization of the speed controller *)
	SimulationModel : MTWinderSimulationModel; (* function block MTWinderSimulationModel *)
END_VAR
(* Axis Controller *)
VAR
	AxisController : MTWinderAxisController;
	SetMaterialTension : REAL := 0.0;
	SynchronistionTime : REAL := 0.0;
	StartSynchronisation : BOOL := FALSE;
	StopSynchronisation : BOOL := FALSE;
	ActInertia : REAL;
END_VAR
```

Listed in the project but not available here: Logical/Axis/VMaster/Exit.st, Logical/Axis/AxisObject/RealAxis/AxInit, Logical/Axis/AxisObject/RealAxis/AcpParTab, Logical/Axis/AxisObject/Virtual, Logical/DancerCtrl/DancerController/Exit.st, Logical/DancerCtrl/DancerController/Types.typ
